PROGRAM MAIN
VAR
END_VAR

END_PROGRAM

(* stored: Version 1.1.0.1
   POU MAIN: Id {5d5aa18d-ea80-45c4-b2c2-54f217a5ac0b} *)
